INTERFACE I_CollectionDisposedEvent EXTENDS I_Event

PROPERTY PUBLIC Target : I_Collection
GET
END_GET
END_PROPERTY

END_INTERFACE

(* stored: Version 1.1.0.1, ProductVersion 3.1.4024.12
   Itf I_CollectionDisposedEvent: Id {cc192627-4512-4bdb-8efd-9fc76204cf06}
   Property Target: Id {9a6a2fc4-0aca-43f7-977a-4839fc2aad50}
   Get Get: Id {735418f0-125e-4002-bc0b-68cd468631fd} *)
